(* IEC 61131-3 sources: volt/packages/volt-lsp-iec/test-corpus/awa-palletizer/Device/Plc Logic/Application/Library Manager/(unresolved)/cmpusermgr interfaces, 13 files *)

(* ---- EVTPARAM_CMPUSERMGRDATABASECHANGED.dut ---- *)
TYPE EVTPARAM_CMPUSERMGRDATABASECHANGED :
STRUCT
	BUSERMANAGEMENTCHANGED : DINT;
	BRIGHTSMANAGEMENTCHANGED : DINT;
END_STRUCT
END_TYPE

(* ---- EVTPARAM_CMPUSERMGRPASSWORDVALIDITY.dut ---- *)
TYPE EVTPARAM_CMPUSERMGRPASSWORDVALIDITY :
STRUCT
	PSZUSER : POINTER TO STRING;
	TSETUTC : ULINT;
	TUNTILUTC : ULINT;
END_STRUCT
END_TYPE

(* ---- USERMGRCACHEVALUE.dut ---- *)
TYPE USERMGRCACHEVALUE :
STRUCT
	TYPECLASS : UserMgrTypeClass;
	VALUE : UserMgrValue;
END_STRUCT
END_TYPE

(* ---- USERMGRCREDENTIALS.dut ---- *)
TYPE USERMGRCREDENTIALS :
STRUCT
	CREDENTIALSTYPE : UserMgrCredentials_Type;
	CREDENTIAL : UserMgrCredentials_Store;
END_STRUCT
END_TYPE

(* ---- USERMGRCREDENTIALS_PASSWORD.dut ---- *)
TYPE USERMGRCREDENTIALS_PASSWORD :
STRUCT
	PSZPASSWORD : POINTER TO STRING;
END_STRUCT
END_TYPE

(* ---- USERMGRCREDENTIALS_STORE.dut ---- *)
TYPE USERMGRCREDENTIALS_STORE :
UNION
	PWD : UserMgrCredentials_Password;
END_UNION
END_TYPE

(* ---- USERMGRCREDENTIALS_TYPE.dut ---- *)
TYPE USERMGRCREDENTIALS_TYPE :
(
	PASSWORD := 1
);
END_TYPE

(* ---- USERMGRTYPECLASS.dut ---- *)
TYPE USERMGRTYPECLASS :
(
	TYPE_I8 := 0,
	TYPE_I16,
	TYPE_I32,
	TYPE_UI8,
	TYPE_UI16,
	TYPE_UI32,
	TYPE_REAL32,
	TYPE_REAL64,
	TYPE_HANDLE,
	TYPE_RESULT,
	TYPE_SIZE,
	TYPE_BOOL,
	TYPE_UI64,
	TYPE_I64,
	TYPE_STRING,
	TYPE_WSTRING
);
END_TYPE

(* ---- USERMGRVALUE.dut ---- *)
TYPE USERMGRVALUE :
UNION
	I8VALUE : SINT;
	I16VALUE : INT;
	I32VALUE : DINT;
	UI8VALUE : USINT;
	UI16VALUE : UINT;
	UI32VALUE : UDINT;
	REAL32VALUE : REAL;
	REAL64VALUE : LREAL;
	HANDLEVALUE : RTS_IEC_HANDLE;
	RESULTVALUE : RTS_IEC_RESULT;
	SIZEVALUE : __XWORD;
	BOOLVALUE : BOOL;
	UI64VALUE : ULINT;
	I64VALUE : LINT;
	STRINGVALUE : POINTER TO STRING;
	WSTRINGVALUE : POINTER TO WSTRING;
END_UNION
END_TYPE

(* ---- AUDITINFOIDS.gvl ---- *)
VAR_GLOBAL
	AUDIT_INFOID_USER_LOCKED : DINT := 16#1;
END_VAR

(* ---- CONSTANTS.gvl ---- *)
VAR_GLOBAL
	USERMGR_RIGHT_NONE : DWORD := 0;
	USERMGR_RIGHT_VIEW : DWORD := 1;
	USERMGR_RIGHT_MODIFY : DWORD := 2;
	USERMGR_RIGHT_EXECUTE : DWORD := 4;
	USERMGR_RIGHT_ADD_REMOVE : DWORD := 8;
	USERMGR_RIGHT_OEM : DWORD := 16#FF000000;
	USERMGR_RIGHT_ALL : DWORD := 16#FFFFFFFF;
END_VAR

(* ---- EVENTIDS.gvl ---- *)
VAR_GLOBAL
	CMPID_CMPUSERMGR : DWORD := 16#61;
	EVTPARAMID_CMPUSERMGRDATABASECHANGED : WORD := 16#1;
	EVTVERSION_CMPUSERMGRDATABASECHANGED : WORD := 16#1;
	EVT_USERMGRDATABASECHANGED : DWORD := (SHL(UINT_TO_DWORD(EVTCLASS_INFO), 16) OR 16#1);
	EVTPARAMID_CMPUSERMGRPASSWORDVALIDITY : WORD := 16#3;
	EVTVERSION_CMPUSERMGRPASSWORDVALIDITY : WORD := 16#1;
	EVT_USERMGRPASSWORDVALIDITY : DWORD := (SHL(UINT_TO_DWORD(EVTCLASS_INFO), 16) OR 16#5);
	EVT_USERMGRPASSWORDEXPIRED : DWORD := (SHL(UINT_TO_DWORD(EVTCLASS_WARNING), 16) OR 16#6);
END_VAR

(* ---- PROPERTIES.gvl ---- *)
VAR_GLOBAL
	USERMGR_USER_PROP_PASSWORD_EXPIRED : DWORD := 16#1000;
	USERMGR_USER_PROP_ALLOW_CHANGE_PASSWORD : DWORD := 16#2000;
	USERMGR_USER_PROP_DEFAULT : DWORD := (USERMGR_USER_PROP_ALLOW_CHANGE_PASSWORD + USERMGR_USER_PROP_PASSWORD_EXPIRED);
END_VAR
